TYPE Fahrenheit EXTENDS TerminalStatus :
STRUCT
    _ : LREAL;
END_STRUCT
END_TYPE

(* stored: Version 1.1.0.1, ProductVersion 3.1.4024.4
   DUT Fahrenheit: Id {a3c852d2-6558-4da1-a321-b016a21ba0b5} *)
